FUNCTION_BLOCK FB_Cell_01 EXTENDS FB_PMLUnit IMPLEMENTS I_UnitState
VAR_INPUT
END_VAR
VAR_OUTPUT
END_VAR
VAR
END_VAR

SUPER^();

A_Alarms();

ACTION A_Alarms:


// probably use the event logger
END_ACTION

{warning 'add method implementation '}
METHOD M_Aborted
END_METHOD

{warning 'add method implementation '}
METHOD M_Aborting
M_StateComplete();
END_METHOD

{warning 'add method implementation '}
METHOD M_Clearing
M_StateComplete();
END_METHOD

{warning 'add method implementation '}
METHOD M_Complete
END_METHOD

{warning 'add method implementation '}
METHOD M_Completing
M_StateComplete();
END_METHOD

{warning 'add method implementation '}
METHOD M_Execute
END_METHOD

{warning 'add method implementation '}
METHOD M_Held
END_METHOD

{warning 'add method implementation '}
METHOD M_Holding
M_StateComplete();
END_METHOD

{warning 'add method implementation '}
METHOD M_Idle
END_METHOD

{warning 'add method implementation '}
METHOD M_Resetting
M_StateComplete();
END_METHOD

{warning 'add method implementation '}
METHOD M_Starting
M_StateComplete();
END_METHOD

{warning 'add method implementation '}
METHOD M_StateComplete
fbPML_StateMachine.M_StateComplete();
END_METHOD

{warning 'add method implementation '}
METHOD M_Stopped
END_METHOD

{warning 'add method implementation '}
METHOD M_Stopping
M_StateComplete();
END_METHOD

{warning 'add method implementation '}
METHOD M_Suspended
END_METHOD

{warning 'add method implementation '}
METHOD M_Suspending
M_StateComplete();
END_METHOD

{warning 'add method implementation '}
METHOD M_Undefined
END_METHOD

{warning 'add method implementation '}
METHOD M_Unholding
M_StateComplete();
END_METHOD

{warning 'add method implementation '}
METHOD M_Unsuspending
M_StateComplete();
END_METHOD

END_FUNCTION_BLOCK

(* stored: Version 1.1.0.1, ProductVersion 3.1.4024.11
   POU FB_Cell_01: Id {f81d340e-7374-46bf-8c87-6674d95ca016}, SpecialFunc None
   Folder PML States: Id {06962f23-4d6b-418d-bb82-d0c3ed8aad1f}
   Folder Unit Code: Id {6389f8c2-4269-40e8-be81-d3a3c96e0ed3}
   Action A_Alarms: Id {f36bf467-742c-4eba-8e0d-06ed3b66da67}
   Method M_Aborted: Id {c2e17ba0-3f79-494a-a672-724788bc56d5}
   Method M_Aborting: Id {5bbd67de-1611-4f4a-8d81-54fb23660d8b}
   Method M_Clearing: Id {524efffa-efc7-40df-bc66-0c496f3a1ad0}
   Method M_Complete: Id {24efea04-723f-4dd4-95be-df21a60c7783}
   Method M_Completing: Id {d20faca9-c23e-4395-93ce-606afa71292a}
   Method M_Execute: Id {51af48d1-812c-4442-9b99-ca8cf3cba270}
   Method M_Held: Id {e9c2e2a1-5f29-4541-b164-b911b335fd5a}
   Method M_Holding: Id {5f63ccc2-86ec-4573-b09d-93c23658e4b4}
   Method M_Idle: Id {656b4abc-8219-4a09-bf4a-83f6aa99c008}
   Method M_Resetting: Id {c4da6461-ac93-4e1e-91ef-38c8cc8ac304}
   Method M_Starting: Id {8b2da4bf-31f8-48a3-b0fc-14e794fc2b8c}
   Method M_StateComplete: Id {f0298424-68c1-464e-b4a1-7f6a3075e434}
   Method M_Stopped: Id {aaed99c7-082f-4121-9a5f-e5843664b3cb}
   Method M_Stopping: Id {2b94f682-ff63-4d8b-a7c6-22a290fcd134}
   Method M_Suspended: Id {0b88f180-1bff-496a-af9c-2a38c2ee9403}
   Method M_Suspending: Id {87355f19-095a-42b8-9a25-c093ee93fae3}
   Method M_Undefined: Id {2943cac7-d462-4df5-a894-c5fdc1b61114}
   Method M_Unholding: Id {5ea4b7e1-59f6-4afc-9188-940cfeb80b88}
   Method M_Unsuspending: Id {64f252e1-2c60-4172-8c46-850e4b06c07c} *)
